FUNCTION_BLOCK ctb2
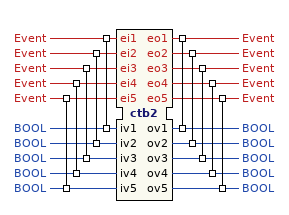
  EVENT_INPUT
    ei1 WITH iv1;
    ei2 WITH iv2;
    ei3 WITH iv3;
    ei4 WITH iv4;
    ei5 WITH iv5;
  END_EVENT
  EVENT_OUTPUT
    eo1 WITH ov1;
    eo2 WITH ov2;
    eo3 WITH ov3;
    eo4 WITH ov4;
    eo5 WITH ov5;
  END_EVENT
  VAR_INPUT
    iv1 : BOOL;
    iv2 : BOOL;
    iv3 : BOOL;
    iv4 : BOOL;
    iv5 : BOOL;
  END_VAR
  VAR_OUTPUT
    ov1 : BOOL;
    ov2 : BOOL;
    ov3 : BOOL;
    ov4 : BOOL;
    ov5 : BOOL;
  END_VAR
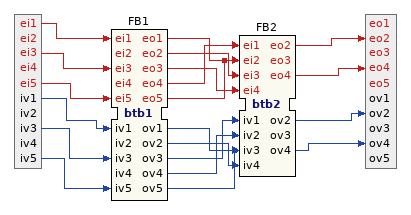
  FBS
    FB1 : btb1;
    FB2 : btb2;
  END_FBS
  EVENT_CONNECTIONS
    ei1 TO FB1.ei1;
    ei3 TO FB1.ei3;
    ei5 TO FB1.ei5;
    FB2.eo2 TO eo2;
    FB2.eo4 TO eo4;
    FB1.eo1 TO FB2.ei2;
    FB1.eo2 TO FB2.ei3;
    FB1.eo3 TO FB2.ei4;
    FB1.eo4 TO FB2.ei1;
    FB1.eo5 TO FB2.ei2;
  END_CONNECTIONS
  DATA_CONNECTIONS
    iv1 TO FB1.iv1;
    iv3 TO FB1.iv3;
    iv5 TO FB1.iv5;
    FB2.ov2 TO ov2;
    FB2.ov4 TO ov4;
    FB1.ov1 TO FB2.iv3;
    FB1.ov2 TO FB2.iv4;
    FB1.ov3 TO FB2.iv1;
    FB1.ov4 TO FB2.iv2;
    FB1.ov5 TO FB2.iv3;
  END_CONNECTIONS
END_FUNCTION_BLOCK
